// TIA Portal V19 export
TYPE "C701_VAR_IF_KMO_TYPIC"
   STRUCT
      STO { ExternalAccessible := 'False'; ExternalVisible := 'False'; ExternalWritable := 'False'} : Struct   // Opsomming van alle storingen
         A001 : Bool;   // Fout temperatuurmeting koelwater in
         A002 : Bool;   // Fout temperatuurmeting koelwater uit
         A003 : Bool;   // Fout drukmeting koelwater
         A004 : Bool;   // Fout flowmeting koelwater
         A005 : Bool;   // Fout algemeen koelmachine
         A006 : Bool;   // Fout circulatiepomp
      END_STRUCT;
   END_STRUCT;
END_TYPE
